// TIA Portal V20 export
DATA_BLOCK "DB_Alarm"   // DB16
// stored: Access Published, MemoryReserve 100, Namespace LineC1
   VAR
      "word" : Struct
         Line : Struct
            C1 : Struct
               Conveyor : Array[_.minC1.._.maxC1] of Word;
            END_STRUCT;
         END_STRUCT;
      END_STRUCT;
   END_VAR
BEGIN
END_DATA_BLOCK
